(* IEC 61131-3 sources: SIMERLIFT/LOGICAD/SIMERLIFT/src_FBD/fbdCommon/Library, 6 files *)

(* ---- DEMUX_2.iecfbd ---- *)
FUNCTION_BLOCK DEMUX_2
  {
    IN {index := 0};
    Select {index := 1};
    OUT_0 {index := 0};
    OUT_1 {index := 1};
    width := 200;
  }

  VAR_INPUT
    Select : BOOL := 0;
    IN : UDINT := 0;
  END_VAR
  VAR_OUTPUT
    OUT_0 : UDINT := 0;
    OUT_1 : UDINT := 0;
  END_VAR

  (*

    // Network 1:
    EQ(IN1 := Select, IN2 := 0, EQ => @C(11).EQ);
    SEL_UDINT(G := @C(11).EQ, IN0 := 0, IN1 := IN, SEL_UDINT => OUT_0);
    EQ(IN1 := Select, IN2 := 1, EQ => @C(14).EQ);
    SEL_UDINT(G := @C(14).EQ, IN0 := 0, IN1 := IN, SEL_UDINT => OUT_1);

  *)

  @VF(1) : @E(Select), @R(20.0, 20.0, 220.0, 19.0);
  @C(11) : @F(EQ), @R(320.0, 20.0, 40.0, 38.0), BOOL, @I(@N(IN1), @L(9.5)), @I(@N(IN2), @L(29.5)), @O(@N(EQ), @R(9.5));
  @C(14) : @F(EQ), @R(320.0, 80.0, 40.0, 38.0), BOOL, @I(@N(IN1), @L(9.5)), @I(@N(IN2), @L(29.5)), @O(@N(EQ), @R(9.5));
  @C(42) : @F(SEL_UDINT), @R(590.0, 20.0, 120.0, 58.0), @I(@N(G), @L(9.5)), @I(@N(IN0), @L(29.5)), @I(@N(IN1), @L(49.5)), @O(@N(SEL_UDINT), @R(9.5));
  @C(48) : @F(SEL_UDINT), @R(590.0, 80.0, 120.0, 58.0), @I(@N(G), @L(9.5)), @I(@N(IN0), @L(29.5)), @I(@N(IN1), @L(49.5)), @O(@N(SEL_UDINT), @R(9.5));
  @VF(185) : @E(0), @R(130.0, 40.0, 110.0, 19.0), BOOL;
  @VF(44) : @E(0), @R(440.0, 40.0, 110.0, 19.0), UDINT;
  @VF(16) : @E(1), @R(130.0, 100.0, 110.0, 19.0), BOOL;
  @VF(50) : @E(0), @R(440.0, 100.0, 110.0, 19.0), UDINT;
  @VF(2) : @E(IN), @R(20.0, 60.0, 220.0, 19.0);
  @VF(5) : @E(OUT_0), @R(750.0, 20.0, 220.0, 19.0);
  @VF(6) : @E(OUT_1), @R(750.0, 80.0, 220.0, 19.0);
  @CP(15) : 279.5, 29.5;
  @CP(4) : 399.5, 69.5;

  @G(12) :
     @L(@CP(15), @C(11).IN1),
     @L(@CP(15), @C(14).IN1),
     @L(@VF(1).o, @CP(15))
    ;
  @G(13) :
     @L(@VF(185).o, @C(11).IN2)
    ;
  @G(43) :
     @L(@C(11).EQ, @C(42).G)
    ;
  @G(45) :
     @L(@VF(44).o, @C(42).IN0)
    ;
  @G(83) :
     @L(@C(14).EQ, @C(48).G)
    ;
  @G(17) :
     @L(@VF(16).o, @C(14).IN2)
    ;
  @G(52) :
     @L(@VF(50).o, @C(48).IN0)
    ;
  @G(3) :
     @L(@VF(2).o, @CP(4)),
     @L(@CP(4), @C(42).IN1),
     @L(@CP(4), @C(48).IN1)
    ;
  @G(7) :
     @L(@C(42).SEL_UDINT, @VF(5).i)
    ;
  @G(8) :
     @L(@C(48).SEL_UDINT, @VF(6).i)
    ;
END_FUNCTION_BLOCK

(* ---- DEMUX_8.iecfbd ---- *)
FUNCTION_BLOCK DEMUX_8
  {
    Select {index := 1};
    OUT_0 {index := 0};
    IN {index := 0};
    OUT_1 {index := 1};
    OUT_2 {index := 2};
    OUT_3 {index := 3};
    OUT_4 {index := 4};
    OUT_5 {index := 5};
    OUT_6 {index := 6};
    OUT_7 {index := 7};
    width := 200;
  }

  VAR_INPUT
    Select : BYTE := 0;
    IN : UDINT := 0;
  END_VAR
  VAR_OUTPUT
    OUT_0 : UDINT := 0;
    OUT_1 : UDINT := 0;
    OUT_2 : UDINT := 0;
    OUT_3 : UDINT := 0;
    OUT_4 : UDINT := 0;
    OUT_5 : UDINT := 0;
    OUT_6 : UDINT := 0;
    OUT_7 : UDINT := 0;
  END_VAR

  (*

    // Network 1:
    EQ(IN1 := Select, IN2 := 0, EQ => @C(11).EQ);
    SEL_UDINT(G := @C(11).EQ, IN0 := 0, IN1 := IN, SEL_UDINT => OUT_0);
    EQ(IN1 := Select, IN2 := 1, EQ => @C(14).EQ);
    SEL_UDINT(G := @C(14).EQ, IN0 := 0, IN1 := IN, SEL_UDINT => OUT_1);
    EQ(IN1 := Select, IN2 := 2, EQ => @C(18).EQ);
    SEL_UDINT(G := @C(18).EQ, IN0 := 0, IN1 := IN, SEL_UDINT => OUT_2);
    EQ(IN1 := Select, IN2 := 3, EQ => @C(21).EQ);
    SEL_UDINT(G := @C(21).EQ, IN0 := 0, IN1 := IN, SEL_UDINT => OUT_3);
    EQ(IN1 := Select, IN2 := 4, EQ => @C(24).EQ);
    SEL_UDINT(G := @C(24).EQ, IN0 := 0, IN1 := IN, SEL_UDINT => OUT_4);
    EQ(IN1 := Select, IN2 := 5, EQ => @C(27).EQ);
    SEL_UDINT(G := @C(27).EQ, IN0 := 0, IN1 := IN, SEL_UDINT => OUT_5);
    EQ(IN1 := Select, IN2 := 6, EQ => @C(30).EQ);
    SEL_UDINT(G := @C(30).EQ, IN0 := 0, IN1 := IN, SEL_UDINT => OUT_6);
    EQ(IN1 := Select, IN2 := 7, EQ => @C(33).EQ);
    SEL_UDINT(G := @C(33).EQ, IN0 := 0, IN1 := IN, SEL_UDINT => OUT_7);

  *)

  @VF(9) : @E(Select), @R(20.0, 20.0, 220.0, 19.0);
  @C(11) : @F(EQ), @R(320.0, 20.0, 40.0, 38.0), BYTE, @I(@N(IN1), @L(9.5)), @I(@N(IN2), @L(29.5)), @O(@N(EQ), @R(9.5));
  @VF(185) : @E(0), @R(130.0, 40.0, 110.0, 19.0), BYTE;
  @C(14) : @F(EQ), @R(320.0, 80.0, 40.0, 38.0), BYTE, @I(@N(IN1), @L(9.5)), @I(@N(IN2), @L(29.5)), @O(@N(EQ), @R(9.5));
  @VF(16) : @E(1), @R(130.0, 100.0, 110.0, 19.0), BYTE;
  @C(18) : @F(EQ), @R(320.0, 140.0, 40.0, 38.0), BYTE, @I(@N(IN1), @L(9.5)), @I(@N(IN2), @L(29.5)), @O(@N(EQ), @R(9.5));
  @VF(19) : @E(2), @R(130.0, 160.0, 110.0, 19.0), BYTE;
  @C(21) : @F(EQ), @R(320.0, 200.0, 40.0, 38.0), BYTE, @I(@N(IN1), @L(9.5)), @I(@N(IN2), @L(29.5)), @O(@N(EQ), @R(9.5));
  @VF(22) : @E(3), @R(130.0, 220.0, 110.0, 19.0), BYTE;
  @C(24) : @F(EQ), @R(320.0, 260.0, 40.0, 38.0), BYTE, @I(@N(IN1), @L(9.5)), @I(@N(IN2), @L(29.5)), @O(@N(EQ), @R(9.5));
  @VF(25) : @E(4), @R(130.0, 280.0, 110.0, 19.0), BYTE;
  @C(27) : @F(EQ), @R(320.0, 320.0, 40.0, 38.0), BYTE, @I(@N(IN1), @L(9.5)), @I(@N(IN2), @L(29.5)), @O(@N(EQ), @R(9.5));
  @VF(28) : @E(5), @R(130.0, 340.0, 110.0, 19.0), BYTE;
  @C(30) : @F(EQ), @R(320.0, 380.0, 40.0, 38.0), BYTE, @I(@N(IN1), @L(9.5)), @I(@N(IN2), @L(29.5)), @O(@N(EQ), @R(9.5));
  @VF(31) : @E(6), @R(130.0, 400.0, 110.0, 19.0), BYTE;
  @C(33) : @F(EQ), @R(320.0, 440.0, 40.0, 38.0), BYTE, @I(@N(IN1), @L(9.5)), @I(@N(IN2), @L(29.5)), @O(@N(EQ), @R(9.5));
  @VF(34) : @E(7), @R(130.0, 460.0, 110.0, 19.0), BYTE;
  @VF(1) : @E(OUT_1), @R(750.0, 80.0, 220.0, 19.0);
  @VF(2) : @E(OUT_2), @R(750.0, 140.0, 220.0, 19.0);
  @VF(3) : @E(OUT_3), @R(750.0, 200.0, 220.0, 19.0);
  @VF(4) : @E(OUT_4), @R(750.0, 260.0, 220.0, 19.0);
  @VF(5) : @E(OUT_5), @R(750.0, 320.0, 220.0, 19.0);
  @VF(6) : @E(OUT_6), @R(750.0, 380.0, 220.0, 19.0);
  @VF(7) : @E(OUT_7), @R(750.0, 440.0, 220.0, 19.0);
  @VF(8) : @E(IN), @R(20.0, 60.0, 220.0, 19.0);
  @C(42) : @F(SEL_UDINT), @R(590.0, 20.0, 120.0, 58.0), @I(@N(G), @L(9.5)), @I(@N(IN0), @L(29.5)), @I(@N(IN1), @L(49.5)), @O(@N(SEL_UDINT), @R(9.5));
  @VF(44) : @E(0), @R(440.0, 40.0, 110.0, 19.0), UDINT;
  @VF(47) : @E(OUT_0), @R(750.0, 20.0, 220.0, 19.0);
  @C(48) : @F(SEL_UDINT), @R(590.0, 80.0, 120.0, 58.0), @I(@N(G), @L(9.5)), @I(@N(IN0), @L(29.5)), @I(@N(IN1), @L(49.5)), @O(@N(SEL_UDINT), @R(9.5));
  @VF(50) : @E(0), @R(440.0, 100.0, 110.0, 19.0), UDINT;
  @C(53) : @F(SEL_UDINT), @R(590.0, 200.0, 120.0, 58.0), @I(@N(G), @L(9.5)), @I(@N(IN0), @L(29.5)), @I(@N(IN1), @L(49.5)), @O(@N(SEL_UDINT), @R(9.5));
  @C(54) : @F(SEL_UDINT), @R(590.0, 140.0, 120.0, 58.0), @I(@N(G), @L(9.5)), @I(@N(IN0), @L(29.5)), @I(@N(IN1), @L(49.5)), @O(@N(SEL_UDINT), @R(9.5));
  @VF(56) : @E(0), @R(440.0, 160.0, 110.0, 19.0), UDINT;
  @VF(58) : @E(0), @R(440.0, 220.0, 110.0, 19.0), UDINT;
  @C(63) : @F(SEL_UDINT), @R(590.0, 440.0, 120.0, 58.0), @I(@N(G), @L(9.5)), @I(@N(IN0), @L(29.5)), @I(@N(IN1), @L(49.5)), @O(@N(SEL_UDINT), @R(9.5));
  @C(64) : @F(SEL_UDINT), @R(590.0, 380.0, 120.0, 58.0), @I(@N(G), @L(9.5)), @I(@N(IN0), @L(29.5)), @I(@N(IN1), @L(49.5)), @O(@N(SEL_UDINT), @R(9.5));
  @C(65) : @F(SEL_UDINT), @R(590.0, 320.0, 120.0, 58.0), @I(@N(G), @L(9.5)), @I(@N(IN0), @L(29.5)), @I(@N(IN1), @L(49.5)), @O(@N(SEL_UDINT), @R(9.5));
  @C(66) : @F(SEL_UDINT), @R(590.0, 260.0, 120.0, 58.0), @I(@N(G), @L(9.5)), @I(@N(IN0), @L(29.5)), @I(@N(IN1), @L(49.5)), @O(@N(SEL_UDINT), @R(9.5));
  @VF(68) : @E(0), @R(440.0, 280.0, 110.0, 19.0), UDINT;
  @VF(70) : @E(0), @R(440.0, 340.0, 110.0, 19.0), UDINT;
  @VF(72) : @E(0), @R(440.0, 400.0, 110.0, 19.0), UDINT;
  @VF(74) : @E(0), @R(440.0, 460.0, 110.0, 19.0), UDINT;
  @CP(15) : 279.5, 29.5;
  @CP(36) : 279.5, 89.5;
  @CP(37) : 279.5, 149.5;
  @CP(38) : 279.5, 209.5;
  @CP(39) : 279.5, 269.5;
  @CP(40) : 279.5, 329.5;
  @CP(41) : 279.5, 389.5;
  @CP(49) : 399.5, 69.5;
  @CP(51) : 399.5, 129.5;
  @CP(55) : 399.5, 189.5;
  @CP(57) : 399.5, 249.5;
  @CP(59) : 399.5, 309.5;
  @CP(61) : 399.5, 369.5;
  @CP(67) : 399.5, 429.5;

  @G(12) :
     @L(@VF(9).o, @CP(15)),
     @L(@CP(15), @C(11).IN1),
     @L(@CP(15), @CP(36)),
     @L(@CP(36), @C(14).IN1),
     @L(@CP(36), @CP(37)),
     @L(@CP(37), @C(18).IN1),
     @L(@CP(37), @CP(38)),
     @L(@CP(38), @C(21).IN1),
     @L(@CP(38), @CP(39)),
     @L(@CP(39), @C(24).IN1),
     @L(@CP(39), @CP(40)),
     @L(@CP(40), @C(27).IN1),
     @L(@CP(40), @CP(41)),
     @L(@CP(41), @C(30).IN1),
     @L(@CP(41), @C(33).IN1)
    ;
  @G(13) :
     @L(@VF(185).o, @C(11).IN2)
    ;
  @G(17) :
     @L(@VF(16).o, @C(14).IN2)
    ;
  @G(20) :
     @L(@VF(19).o, @C(18).IN2)
    ;
  @G(23) :
     @L(@VF(22).o, @C(21).IN2)
    ;
  @G(26) :
     @L(@VF(25).o, @C(24).IN2)
    ;
  @G(29) :
     @L(@VF(28).o, @C(27).IN2)
    ;
  @G(32) :
     @L(@VF(31).o, @C(30).IN2)
    ;
  @G(35) :
     @L(@VF(34).o, @C(33).IN2)
    ;
  @G(43) :
     @L(@C(11).EQ, @C(42).G)
    ;
  @G(45) :
     @L(@VF(44).o, @C(42).IN0)
    ;
  @G(46) :
     @L(@VF(8).o, @CP(49)),
     @L(@CP(49), @C(42).IN1),
     @L(@CP(49), @CP(51)),
     @L(@CP(51), @C(48).IN1),
     @L(@CP(51), @CP(55)),
     @L(@CP(55), @C(54).IN1),
     @L(@CP(55), @CP(57)),
     @L(@CP(57), @C(53).IN1),
     @L(@CP(57), @CP(59)),
     @L(@CP(59), @C(66).IN1),
     @L(@CP(59), @CP(61)),
     @L(@CP(61), @C(65).IN1),
     @L(@CP(61), @CP(67)),
     @L(@CP(67), @C(64).IN1),
     @L(@CP(67), @C(63).IN1)
    ;
  @G(10) :
     @L(@C(42).SEL_UDINT, @VF(47).i)
    ;
  @G(52) :
     @L(@VF(50).o, @C(48).IN0)
    ;
  @G(60) :
     @L(@VF(58).o, @C(53).IN0)
    ;
  @G(62) :
     @L(@VF(56).o, @C(54).IN0)
    ;
  @G(77) :
     @L(@VF(74).o, @C(63).IN0)
    ;
  @G(79) :
     @L(@VF(72).o, @C(64).IN0)
    ;
  @G(80) :
     @L(@VF(70).o, @C(65).IN0)
    ;
  @G(82) :
     @L(@VF(68).o, @C(66).IN0)
    ;
  @G(83) :
     @L(@C(14).EQ, @C(48).G)
    ;
  @G(84) :
     @L(@C(18).EQ, @C(54).G)
    ;
  @G(85) :
     @L(@C(21).EQ, @C(53).G)
    ;
  @G(86) :
     @L(@C(24).EQ, @C(66).G)
    ;
  @G(87) :
     @L(@C(27).EQ, @C(65).G)
    ;
  @G(88) :
     @L(@C(30).EQ, @C(64).G)
    ;
  @G(89) :
     @L(@C(33).EQ, @C(63).G)
    ;
  @G(90) :
     @L(@C(48).SEL_UDINT, @VF(1).i)
    ;
  @G(91) :
     @L(@C(54).SEL_UDINT, @VF(2).i)
    ;
  @G(92) :
     @L(@C(53).SEL_UDINT, @VF(3).i)
    ;
  @G(93) :
     @L(@C(66).SEL_UDINT, @VF(4).i)
    ;
  @G(94) :
     @L(@C(65).SEL_UDINT, @VF(5).i)
    ;
  @G(95) :
     @L(@C(64).SEL_UDINT, @VF(6).i)
    ;
  @G(96) :
     @L(@C(63).SEL_UDINT, @VF(7).i)
    ;
END_FUNCTION_BLOCK

(* ---- Select_12.iecfbd ---- *)
FUNCTION_BLOCK Select_12
  {
    In00 {index := 0};
    In01 {index := 2};
    In02 {index := 4};
    In03 {index := 6};
    In04 {index := 8};
    In05 {index := 10};
    In06 {index := 12};
    In07 {index := 14};
    S00 {index := 1};
    S01 {index := 3};
    S02 {index := 5};
    S03 {index := 7};
    S04 {index := 9};
    S05 {index := 11};
    S06 {index := 13};
    In08 {index := 16};
    In09 {index := 18};
    In10 {index := 20};
    In11 {index := 22};
    S07 {index := 15};
    S08 {index := 17};
    S09 {index := 19};
    S10 {index := 21};
    S11 {index := 23};
    i {index := 25};
    Q {index := 0};
    width := 160;
    height := 518;
  }

  VAR_INPUT
    In00 : WORD := 0;
    In01 : WORD := 0;
    In02 : WORD := 0;
    In03 : WORD := 0;
    In04 : WORD := 0;
    In05 : WORD := 0;
    In06 : WORD := 0;
    In07 : WORD := 0;
    S00 : BOOL := 0;
    S01 : BOOL := 0;
    S02 : BOOL := 0;
    S03 : BOOL := 0;
    S04 : BOOL := 0;
    S05 : BOOL := 0;
    S06 : BOOL := 0;
    i : BYTE := 0;
    S07 : BOOL := 0;
    In08 : WORD := 0;
    In09 : WORD := 0;
    In10 : WORD := 0;
    In11 : WORD := 0;
    S08 : BOOL := 0;
    S09 : BOOL := 0;
    S10 : BOOL := 0;
    S11 : BOOL := 0;
  END_VAR
  VAR_OUTPUT
    Q : WORD := 0;
  END_VAR

  (*

    // Network 1:
    SEL_WORD(G := S00, IN0 := i, IN1 := In00, SEL_WORD => @C(19).SEL_WORD);
    SEL_WORD(G := S01, IN0 := @C(19).SEL_WORD, IN1 := In01, SEL_WORD => @C(22).SEL_WORD);
    SEL_WORD(G := S02, IN0 := @C(22).SEL_WORD, IN1 := In02, SEL_WORD => @C(24).SEL_WORD);
    SEL_WORD(G := S03, IN0 := @C(24).SEL_WORD, IN1 := In03, SEL_WORD => @C(26).SEL_WORD);
    SEL_WORD(G := S04, IN0 := @C(26).SEL_WORD, IN1 := In04, SEL_WORD => @C(25).SEL_WORD);
    SEL_WORD(G := S05, IN0 := @C(25).SEL_WORD, IN1 := In05, SEL_WORD => @C(28).SEL_WORD);
    SEL_WORD(G := S06, IN0 := @C(28).SEL_WORD, IN1 := In06, SEL_WORD => @C(27).SEL_WORD);
    SEL_WORD(G := S07, IN0 := @C(27).SEL_WORD, IN1 := In07, SEL_WORD => @C(23).SEL_WORD);
    SEL_WORD(G := S08, IN0 := @C(23).SEL_WORD, IN1 := In08, SEL_WORD => @C(54).SEL_WORD);
    SEL_WORD(G := S09, IN0 := @C(54).SEL_WORD, IN1 := In09, SEL_WORD => @C(53).SEL_WORD);
    SEL_WORD(G := S10, IN0 := @C(53).SEL_WORD, IN1 := In10, SEL_WORD => @C(52).SEL_WORD);
    SEL_WORD(G := S11, IN0 := @C(52).SEL_WORD, IN1 := In11, SEL_WORD => Q);

  *)

  @C(19) : @F(SEL_WORD), @R(130.0, 700.0, 120.0, 58.0), @I(@N(G), @L(9.5)), @I(@N(IN0), @L(29.5)), @I(@N(IN1), @L(49.5)), @O(@N(SEL_WORD), @R(9.5));
  @C(23) : @F(SEL_WORD), @R(1110.0, 280.0, 120.0, 58.0), @I(@N(G), @L(9.5)), @I(@N(IN0), @L(29.5)), @I(@N(IN1), @L(49.5)), @O(@N(SEL_WORD), @R(9.5));
  @C(22) : @F(SEL_WORD), @R(270.0, 640.0, 120.0, 58.0), @I(@N(G), @L(9.5)), @I(@N(IN0), @L(29.5)), @I(@N(IN1), @L(49.5)), @O(@N(SEL_WORD), @R(9.5));
  @C(25) : @F(SEL_WORD), @R(690.0, 460.0, 120.0, 58.0), @I(@N(G), @L(9.5)), @I(@N(IN0), @L(29.5)), @I(@N(IN1), @L(49.5)), @O(@N(SEL_WORD), @R(9.5));
  @C(24) : @F(SEL_WORD), @R(410.0, 580.0, 120.0, 58.0), @I(@N(G), @L(9.5)), @I(@N(IN0), @L(29.5)), @I(@N(IN1), @L(49.5)), @O(@N(SEL_WORD), @R(9.5));
  @C(27) : @F(SEL_WORD), @R(970.0, 340.0, 120.0, 58.0), @I(@N(G), @L(9.5)), @I(@N(IN0), @L(29.5)), @I(@N(IN1), @L(49.5)), @O(@N(SEL_WORD), @R(9.5));
  @C(26) : @F(SEL_WORD), @R(550.0, 520.0, 120.0, 58.0), @I(@N(G), @L(9.5)), @I(@N(IN0), @L(29.5)), @I(@N(IN1), @L(49.5)), @O(@N(SEL_WORD), @R(9.5));
  @C(28) : @F(SEL_WORD), @R(830.0, 400.0, 120.0, 58.0), @I(@N(G), @L(9.5)), @I(@N(IN0), @L(29.5)), @I(@N(IN1), @L(49.5)), @O(@N(SEL_WORD), @R(9.5));
  @VF(1) : @E(In00), @R(40.0, 740.0, 70.0, 19.0);
  @VF(2) : @E(In01), @R(40.0, 680.0, 70.0, 19.0);
  @VF(3) : @E(In02), @R(40.0, 620.0, 70.0, 19.0);
  @VF(4) : @E(In03), @R(40.0, 560.0, 70.0, 19.0);
  @VF(5) : @E(In04), @R(40.0, 500.0, 70.0, 19.0);
  @VF(6) : @E(In05), @R(40.0, 440.0, 70.0, 19.0);
  @VF(7) : @E(In06), @R(40.0, 380.0, 70.0, 19.0);
  @VF(8) : @E(In07), @R(40.0, 320.0, 70.0, 19.0);
  @VF(9) : @E(S00), @R(40.0, 700.0, 70.0, 19.0);
  @VF(10) : @E(S01), @R(40.0, 640.0, 70.0, 19.0);
  @VF(11) : @E(S02), @R(40.0, 580.0, 70.0, 19.0);
  @VF(12) : @E(S03), @R(40.0, 520.0, 70.0, 19.0);
  @VF(13) : @E(S04), @R(40.0, 460.0, 70.0, 19.0);
  @VF(14) : @E(S05), @R(40.0, 400.0, 70.0, 19.0);
  @VF(15) : @E(S06), @R(40.0, 340.0, 70.0, 19.0);
  @VF(17) : @E(i), @R(40.0, 720.0, 70.0, 19.0);
  @VF(16) : @E(S07), @R(40.0, 280.0, 70.0, 19.0);
  @C(51) : @F(SEL_WORD), @R(1670.0, 40.0, 120.0, 58.0), @I(@N(G), @L(9.5)), @I(@N(IN0), @L(29.5)), @I(@N(IN1), @L(49.5)), @O(@N(SEL_WORD), @R(9.5));
  @C(52) : @F(SEL_WORD), @R(1530.0, 100.0, 120.0, 58.0), @I(@N(G), @L(9.5)), @I(@N(IN0), @L(29.5)), @I(@N(IN1), @L(49.5)), @O(@N(SEL_WORD), @R(9.5));
  @C(53) : @F(SEL_WORD), @R(1390.0, 160.0, 120.0, 58.0), @I(@N(G), @L(9.5)), @I(@N(IN0), @L(29.5)), @I(@N(IN1), @L(49.5)), @O(@N(SEL_WORD), @R(9.5));
  @C(54) : @F(SEL_WORD), @R(1250.0, 220.0, 120.0, 58.0), @I(@N(G), @L(9.5)), @I(@N(IN0), @L(29.5)), @I(@N(IN1), @L(49.5)), @O(@N(SEL_WORD), @R(9.5));
  @VF(58) : @E(Q), @R(1810.0, 40.0, 70.0, 19.0);
  @VF(18) : @E(In08), @R(40.0, 260.0, 70.0, 19.0);
  @VF(59) : @E(In09), @R(40.0, 200.0, 70.0, 19.0);
  @VF(60) : @E(In10), @R(40.0, 140.0, 70.0, 19.0);
  @VF(61) : @E(In11), @R(40.0, 80.0, 70.0, 19.0);
  @VF(62) : @E(S08), @R(40.0, 220.0, 70.0, 19.0);
  @VF(63) : @E(S09), @R(40.0, 160.0, 70.0, 19.0);
  @VF(64) : @E(S10), @R(40.0, 100.0, 70.0, 19.0);
  @VF(65) : @E(S11), @R(40.0, 40.0, 70.0, 19.0);

  @G(20) :
     @L(@VF(9).o, @C(19).G)
    ;
  @G(21) :
     @L(@VF(1).o, @C(19).IN1)
    ;
  @G(29) :
     @L(@VF(10).o, @C(22).G)
    ;
  @G(30) :
     @L(@VF(11).o, @C(24).G)
    ;
  @G(31) :
     @L(@VF(15).o, @C(27).G)
    ;
  @G(32) :
     @L(@VF(14).o, @C(28).G)
    ;
  @G(33) :
     @L(@VF(13).o, @C(25).G)
    ;
  @G(34) :
     @L(@VF(12).o, @C(26).G)
    ;
  @G(35) :
     @L(@VF(16).o, @C(23).G)
    ;
  @G(36) :
     @L(@VF(2).o, @C(22).IN1)
    ;
  @G(37) :
     @L(@VF(3).o, @C(24).IN1)
    ;
  @G(38) :
     @L(@VF(4).o, @C(26).IN1)
    ;
  @G(39) :
     @L(@VF(5).o, @C(25).IN1)
    ;
  @G(40) :
     @L(@VF(6).o, @C(28).IN1)
    ;
  @G(41) :
     @L(@VF(7).o, @C(27).IN1)
    ;
  @G(42) :
     @L(@VF(8).o, @C(23).IN1)
    ;
  @G(101) :
     @L(@VF(17).o, @C(19).IN0)
    ;
  @G(43) :
     @L(@C(19).SEL_WORD, @C(22).IN0)
    ;
  @G(44) :
     @L(@C(22).SEL_WORD, @C(24).IN0)
    ;
  @G(45) :
     @L(@C(24).SEL_WORD, @C(26).IN0)
    ;
  @G(46) :
     @L(@C(26).SEL_WORD, @C(25).IN0)
    ;
  @G(47) :
     @L(@C(25).SEL_WORD, @C(28).IN0)
    ;
  @G(48) :
     @L(@C(28).SEL_WORD, @C(27).IN0)
    ;
  @G(49) :
     @L(@C(27).SEL_WORD, @C(23).IN0)
    ;
  @G(55) :
     @L(@C(52).SEL_WORD, @C(51).IN0)
    ;
  @G(56) :
     @L(@C(53).SEL_WORD, @C(52).IN0)
    ;
  @G(57) :
     @L(@C(54).SEL_WORD, @C(53).IN0)
    ;
  @G(50) :
     @L(@C(23).SEL_WORD, @C(54).IN0)
    ;
  @G(66) :
     @L(@C(51).SEL_WORD, @VF(58).i)
    ;
  @G(67) :
     @L(@VF(62).o, @C(54).G)
    ;
  @G(68) :
     @L(@VF(63).o, @C(53).G)
    ;
  @G(69) :
     @L(@VF(64).o, @C(52).G)
    ;
  @G(70) :
     @L(@VF(65).o, @C(51).G)
    ;
  @G(71) :
     @L(@VF(61).o, @C(51).IN1)
    ;
  @G(72) :
     @L(@VF(60).o, @C(52).IN1)
    ;
  @G(73) :
     @L(@VF(59).o, @C(53).IN1)
    ;
  @G(74) :
     @L(@VF(18).o, @C(54).IN1)
    ;
END_FUNCTION_BLOCK

(* ---- Select_8.iecfbd ---- *)
FUNCTION_BLOCK Select_8
  {
    In0 {index := 0};
    S0 {index := 1};
    In1 {index := 2};
    S1 {index := 3};
    In2 {index := 4};
    In3 {index := 6};
    In4 {index := 8};
    In5 {index := 10};
    In6 {index := 12};
    In7 {index := 14};
    S2 {index := 5};
    S3 {index := 7};
    S4 {index := 9};
    S5 {index := 11};
    S6 {index := 13};
    S7 {index := 15};
    i {index := 17};
    Q {index := 0};
    width := 160;
    height := 358;
  }

  VAR_INPUT
    In0 : WORD := 0;
    In1 : WORD := 0;
    In2 : WORD := 0;
    In3 : WORD := 0;
    In4 : WORD := 0;
    In5 : WORD := 0;
    In6 : WORD := 0;
    In7 : WORD := 0;
    S0 : BOOL := 0;
    S1 : BOOL := 0;
    S2 : BOOL := 0;
    S3 : BOOL := 0;
    S4 : BOOL := 0;
    S5 : BOOL := 0;
    S6 : BOOL := 0;
    S7 : BOOL := 0;
    i : BYTE := 0;
  END_VAR
  VAR_OUTPUT
    Q : WORD := 0;
  END_VAR

  (*

    // Network 1:
    SEL_WORD(G := S0, IN0 := i, IN1 := In0, SEL_WORD => @C(19).SEL_WORD);
    SEL_WORD(G := S1, IN0 := @C(19).SEL_WORD, IN1 := In1, SEL_WORD => @C(22).SEL_WORD);
    SEL_WORD(G := S2, IN0 := @C(22).SEL_WORD, IN1 := In2, SEL_WORD => @C(24).SEL_WORD);
    SEL_WORD(G := S3, IN0 := @C(24).SEL_WORD, IN1 := In3, SEL_WORD => @C(26).SEL_WORD);
    SEL_WORD(G := S4, IN0 := @C(26).SEL_WORD, IN1 := In4, SEL_WORD => @C(25).SEL_WORD);
    SEL_WORD(G := S5, IN0 := @C(25).SEL_WORD, IN1 := In5, SEL_WORD => @C(28).SEL_WORD);
    SEL_WORD(G := S6, IN0 := @C(28).SEL_WORD, IN1 := In6, SEL_WORD => @C(27).SEL_WORD);
    SEL_WORD(G := S7, IN0 := @C(27).SEL_WORD, IN1 := In7, SEL_WORD => Q);

  *)

  @VF(1) : @E(In0), @R(40.0, 500.0, 140.0, 19.0);
  @VF(2) : @E(In1), @R(40.0, 440.0, 140.0, 19.0);
  @VF(3) : @E(In2), @R(40.0, 380.0, 140.0, 19.0);
  @VF(4) : @E(In3), @R(40.0, 320.0, 140.0, 19.0);
  @VF(5) : @E(In4), @R(40.0, 260.0, 140.0, 19.0);
  @VF(6) : @E(In5), @R(40.0, 200.0, 140.0, 19.0);
  @VF(7) : @E(In6), @R(40.0, 140.0, 140.0, 19.0);
  @VF(8) : @E(In7), @R(40.0, 80.0, 140.0, 19.0);
  @VF(9) : @E(S0), @R(40.0, 460.0, 140.0, 19.0);
  @VF(10) : @E(S1), @R(40.0, 400.0, 140.0, 19.0);
  @VF(11) : @E(S2), @R(40.0, 340.0, 140.0, 19.0);
  @VF(12) : @E(S3), @R(40.0, 280.0, 140.0, 19.0);
  @VF(13) : @E(S4), @R(40.0, 220.0, 140.0, 19.0);
  @VF(14) : @E(S5), @R(40.0, 160.0, 140.0, 19.0);
  @VF(15) : @E(S6), @R(40.0, 100.0, 140.0, 19.0);
  @VF(16) : @E(S7), @R(40.0, 40.0, 140.0, 19.0);
  @VF(17) : @E(i), @R(40.0, 480.0, 140.0, 19.0);
  @VF(18) : @E(Q), @R(1510.0, 40.0, 140.0, 19.0);
  @C(19) : @F(SEL_WORD), @R(220.0, 460.0, 120.0, 58.0), @I(@N(G), @L(9.5)), @I(@N(IN0), @L(29.5)), @I(@N(IN1), @L(49.5)), @O(@N(SEL_WORD), @R(9.5));
  @C(22) : @F(SEL_WORD), @R(380.0, 400.0, 120.0, 58.0), @I(@N(G), @L(9.5)), @I(@N(IN0), @L(29.5)), @I(@N(IN1), @L(49.5)), @O(@N(SEL_WORD), @R(9.5));
  @C(23) : @F(SEL_WORD), @R(1350.0, 40.0, 120.0, 58.0), @I(@N(G), @L(9.5)), @I(@N(IN0), @L(29.5)), @I(@N(IN1), @L(49.5)), @O(@N(SEL_WORD), @R(9.5));
  @C(24) : @F(SEL_WORD), @R(540.0, 340.0, 120.0, 58.0), @I(@N(G), @L(9.5)), @I(@N(IN0), @L(29.5)), @I(@N(IN1), @L(49.5)), @O(@N(SEL_WORD), @R(9.5));
  @C(25) : @F(SEL_WORD), @R(860.0, 220.0, 120.0, 58.0), @I(@N(G), @L(9.5)), @I(@N(IN0), @L(29.5)), @I(@N(IN1), @L(49.5)), @O(@N(SEL_WORD), @R(9.5));
  @C(26) : @F(SEL_WORD), @R(700.0, 280.0, 120.0, 58.0), @I(@N(G), @L(9.5)), @I(@N(IN0), @L(29.5)), @I(@N(IN1), @L(49.5)), @O(@N(SEL_WORD), @R(9.5));
  @C(27) : @F(SEL_WORD), @R(1190.0, 100.0, 120.0, 58.0), @I(@N(G), @L(9.5)), @I(@N(IN0), @L(29.5)), @I(@N(IN1), @L(49.5)), @O(@N(SEL_WORD), @R(9.5));
  @C(28) : @F(SEL_WORD), @R(1030.0, 160.0, 120.0, 58.0), @I(@N(G), @L(9.5)), @I(@N(IN0), @L(29.5)), @I(@N(IN1), @L(49.5)), @O(@N(SEL_WORD), @R(9.5));

  @G(20) :
     @L(@VF(9).o, @C(19).G)
    ;
  @G(21) :
     @L(@VF(1).o, @C(19).IN1)
    ;
  @G(29) :
     @L(@VF(10).o, @C(22).G)
    ;
  @G(30) :
     @L(@VF(11).o, @C(24).G)
    ;
  @G(31) :
     @L(@VF(15).o, @C(27).G)
    ;
  @G(32) :
     @L(@VF(14).o, @C(28).G)
    ;
  @G(33) :
     @L(@VF(13).o, @C(25).G)
    ;
  @G(34) :
     @L(@VF(12).o, @C(26).G)
    ;
  @G(35) :
     @L(@VF(16).o, @C(23).G)
    ;
  @G(36) :
     @L(@VF(2).o, @C(22).IN1)
    ;
  @G(37) :
     @L(@VF(3).o, @C(24).IN1)
    ;
  @G(38) :
     @L(@VF(4).o, @C(26).IN1)
    ;
  @G(39) :
     @L(@VF(5).o, @C(25).IN1)
    ;
  @G(40) :
     @L(@VF(6).o, @C(28).IN1)
    ;
  @G(41) :
     @L(@VF(7).o, @C(27).IN1)
    ;
  @G(42) :
     @L(@VF(8).o, @C(23).IN1)
    ;
  @G(101) :
     @L(@VF(17).o, @C(19).IN0)
    ;
  @G(43) :
     @L(@C(19).SEL_WORD, @C(22).IN0)
    ;
  @G(44) :
     @L(@C(22).SEL_WORD, @C(24).IN0)
    ;
  @G(45) :
     @L(@C(24).SEL_WORD, @C(26).IN0)
    ;
  @G(46) :
     @L(@C(26).SEL_WORD, @C(25).IN0)
    ;
  @G(47) :
     @L(@C(25).SEL_WORD, @C(28).IN0)
    ;
  @G(48) :
     @L(@C(28).SEL_WORD, @C(27).IN0)
    ;
  @G(49) :
     @L(@C(27).SEL_WORD, @C(23).IN0)
    ;
  @G(50) :
     @L(@C(23).SEL_WORD, @VF(18).i)
    ;
END_FUNCTION_BLOCK

(* ---- Temp_CAN.iecfbd ---- *)
FUNCTION_BLOCK Temp_CAN
  {
    Temp {index := 0};
    CAN {index := 0};
    width := 200;
    height := 18;
  }

  VAR
    Lineer_Function1 : Lineer_Function;
  END_VAR
  VAR_INPUT
    Temp : REAL := 0;
  END_VAR
  VAR_OUTPUT
    CAN : USINT := 0;
  END_VAR

  (*

    // Network 1:
    Lineer_Function1(Input := Temp, X1 := -40, X2 := 210, Y1 := 0, Y2 := 250);
    TO_USINT(IN := Lineer_Function1.Lim_Output, TO_USINT => CAN);

  *)

  @VF(1) : @E(Temp), @R(20.0, 40.0, 220.0, 19.0);
  @C(2) : @F(TO_USINT), @R(670.0, 60.0, 120.0, 18.0), LREAL, @I(@N(IN), @L(9.5)), @O(@N(TO_USINT), @R(9.5));
  @C(99) : @FB(Lineer_Function1), @R(430.0, 40.0, 200.0, 118.0), @I(@N(Input), @L(9.5)), @I(@N(X1), @L(29.5)), @I(@N(X2), @L(49.5)), @I(@N(Y1), @L(89.5)), @I(@N(Y2), @L(109.5)), @O(@N(Output), @R(9.5)), @O(@N(Error), @R(109.5)), @O(@N(Lim_Output), @R(29.5));
  @VF(186) : @E(0), @R(280.0, 120.0, 110.0, 19.0), LREAL;
  @VF(188) : @E(250), @R(280.0, 140.0, 110.0, 19.0), LREAL;
  @VF(5) : @E(-40), @R(280.0, 60.0, 110.0, 19.0), LREAL;
  @VF(6) : @E(210), @R(280.0, 80.0, 110.0, 19.0), LREAL;
  @VF(9) : @E(CAN), @R(830.0, 60.0, 220.0, 19.0);

  @G(179) :
     @L(@VF(186).o, @C(99).Y1)
    ;
  @G(187) :
     @L(@VF(188).o, @C(99).Y2)
    ;
  @G(3) :
     @L(@C(99).Lim_Output, @C(2).IN)
    ;
  @G(4) :
     @L(@VF(1).o, @C(99).Input)
    ;
  @G(7) :
     @L(@VF(5).o, @C(99).X1)
    ;
  @G(8) :
     @L(@VF(6).o, @C(99).X2)
    ;
  @G(10) :
     @L(@C(2).TO_USINT, @VF(9).i)
    ;
END_FUNCTION_BLOCK

(* ---- Timer.iecfbd ---- *)
FUNCTION_BLOCK Timer
  {
    T_L {index := 2};
    T_H {index := 1};
    T_Q {index := 1};
    Enable {index := 0};
    Pulse {index := 3};
    P_Q {index := 3};
    width := 120;
    height := 38;
  }

  VAR
    TON4 : TON;
    TON3 : TON;
    TON5 : TON;
    TON6 : TON;
  END_VAR
  VAR_INPUT
    T_H : TIME := T#100ms;
    T_L : TIME := T#100ms;
    Enable : BOOL := 0;
    Pulse : TIME := T#100ms;
  END_VAR
  VAR_OUTPUT
    T_Q : BOOL;
    P_Q : BOOL := 0;
  END_VAR

  (*

    // Network 1:
    DIV_TIME(IN1 := Pulse, IN2 := 2, DIV_TIME => @C(64).DIV_TIME);
    TON4(IN := TON3.Q, PT := T_H);
    NOT(IN := TON4.Q, NOT => @C(33).NOT);
    AND(IN1 := Enable, IN2 := @C(33).NOT, AND => @C(34).AND);
    TON3(IN := @C(34).AND, PT := T_L, Q => T_Q);
    TON6(IN := TON5.Q, PT := @C(64).DIV_TIME);
    NOT(IN := TON6.Q, NOT => @C(62).NOT);
    AND(IN1 := Enable, IN2 := @C(62).NOT, AND => @C(63).AND);
    TON5(IN := @C(63).AND, PT := @C(64).DIV_TIME, Q => P_Q);

  *)

  @C(29) : @FB(TON4), @R(560.0, 100.0, 100.0, 38.0), @I(@N(IN), @L(9.5)), @I(@N(PT), @L(29.5)), @O(@N(Q), @R(9.5)), @O(@N(ET), @R(29.5));
  @C(33) : @F(NOT), @R(160.0, 60.0, 60.0, 18.0), BOOL, @I(@N(IN), @L(9.5)), @O(@N(NOT), @R(9.5));
  @C(34) : @F(AND), @R(260.0, 40.0, 40.0, 38.0), BOOL, @I(@N(IN1), @L(9.5)), @I(@N(IN2), @L(29.5)), @O(@N(AND), @R(9.5));
  @C(37) : @FB(TON3), @R(380.0, 40.0, 100.0, 38.0), @I(@N(IN), @L(9.5)), @I(@N(PT), @L(29.5)), @O(@N(Q), @R(9.5)), @O(@N(ET), @R(29.5));
  @VF(57) : @E(Enable), @R(20.0, 40.0, 200.0, 19.0);
  @VF(59) : @E(P_Q), @R(560.0, 160.0, 200.0, 19.0);
  @C(62) : @F(NOT), @R(160.0, 180.0, 60.0, 18.0), BOOL, @I(@N(IN), @L(9.5)), @O(@N(NOT), @R(9.5));
  @C(63) : @F(AND), @R(260.0, 160.0, 40.0, 38.0), BOOL, @I(@N(IN1), @L(9.5)), @I(@N(IN2), @L(29.5)), @O(@N(AND), @R(9.5));
  @C(64) : @F(DIV_TIME), @R(160.0, 240.0, 40.0, 38.0), USINT, @I(@N(IN1), @L(9.5)), @I(@N(IN2), @L(29.5)), @O(@N(DIV_TIME), @R(9.5));
  @C(65) : @FB(TON5), @R(380.0, 160.0, 100.0, 38.0), @I(@N(IN), @L(9.5)), @I(@N(PT), @L(29.5)), @O(@N(Q), @R(9.5)), @O(@N(ET), @R(29.5));
  @C(66) : @FB(TON6), @R(560.0, 220.0, 100.0, 38.0), @I(@N(IN), @L(9.5)), @I(@N(PT), @L(29.5)), @O(@N(Q), @R(9.5)), @O(@N(ET), @R(29.5));
  @VF(67) : @E(Pulse), @R(20.0, 240.0, 100.0, 19.0);
  @VF(68) : @E(2), @R(20.0, 260.0, 100.0, 19.0), USINT;
  @VF(79) : @E(T_Q), @R(560.0, 40.0, 200.0, 19.0);
  @VF(25) : @E(T_H), @R(20.0, 120.0, 100.0, 19.0);
  @VF(39) : @E(T_L), @R(20.0, 100.0, 100.0, 19.0);
  @CP(43) : 519.5, 49.5;
  @CP(70) : 519.5, 169.5;
  @CP(58) : 239.5, 49.5;
  @CP(9) : 339.5, 249.5;

  @G(51) :
     @L(@C(33).NOT, @C(34).IN2)
    ;
  @G(54) :
     @L(@C(29).Q, @C(33).IN)
    ;
  @G(55) :
     @L(@C(34).AND, @C(37).IN)
    ;
  @G(56) :
     @L(@C(37).Q, @CP(43)),
     @L(@CP(43), @C(29).IN),
     @L(@CP(43), @VF(79).i)
    ;
  @G(71) :
     @L(@C(62).NOT, @C(63).IN2)
    ;
  @G(72) :
     @L(@C(63).AND, @C(65).IN)
    ;
  @G(74) :
     @L(@VF(67).o, @C(64).IN1)
    ;
  @G(75) :
     @L(@VF(68).o, @C(64).IN2)
    ;
  @G(76) :
     @L(@C(65).Q, @CP(70)),
     @L(@CP(70), @C(66).IN),
     @L(@CP(70), @VF(59).i)
    ;
  @G(77) :
     @L(@C(66).Q, @C(62).IN)
    ;
  @G(42) :
     @L(@VF(25).o, @C(29).PT)
    ;
  @G(45) :
     @L(@VF(39).o, @C(37).PT)
    ;
  @G(50) :
     @L(@VF(57).o, @CP(58)),
     @L(@CP(58), @C(34).IN1),
     @L(@CP(58), @C(63).IN1)
    ;
  @G(4) :
     @L(@C(64).DIV_TIME, @CP(9)),
     @L(@CP(9), @C(66).PT),
     @L(@CP(9), @C(65).PT)
    ;
END_FUNCTION_BLOCK
